// TIA Portal V17 export
// export: Created 2025-03-07T09:17:39.7845151Z, ExportSetting WithDefaults, DisplayName Totally Integrated Automation Portal, DisplayVersion V17 Update 8, DisplayName TIA Portal Openness, DisplayVersion V17 Update 8, DisplayName TIA Portal Version Control Interface, DisplayVersion V17, DisplayName SINAMICS Startdrive Advanced, DisplayVersion V17 SP2, DisplayName SINAMICS Startdrive G110M, G120, G120C, G120D, G120P, G115D, DisplayVersion V17 SP2, DisplayName SINAMICS Startdrive G130, G150, S120, S150, SINAMICS MV, S210, DisplayVersion V17 SP2, DisplayName STEP 7 Professional, DisplayVersion V17 Update 8, DisplayName SINUMERIK ONE STEP 7 Toolbox, DisplayVersion V17 Update 12, DisplayName SINUMERIK 840D sl STEP 7 Toolbox, DisplayVersion V17 Update 12, DisplayName STEP 7 Safety, DisplayVersion V17 Update 6, DisplayName WinCC Advanced, DisplayVersion V17 Update 8
FUNCTION "FC2001_AUTO_SINGLE_SEMI_MANUAL" : Void   // FC2001, LAD
{ S7_Optimized_Access := 'FALSE' }
AUTHOR : ETXETAR
VERSION : 1.0
// stored: AutoNumber false, IsIECCheckEnabled false, SetENOAutomatically false, UDAEnableTagReadback false
   VAR_TEMP
      O_BYTE_0 : Struct   // OPTIONS BYTE 0
         CHANGE_MODE_SEOC_ALARM : Bool;   // CHANGE MODE SEOC ALARM OPTION
         MODE_SELECTED_MEMORY : Bool;   // MODE SELECTED MEMORY OPTION
      END_STRUCT;
   END_VAR
   VAR CONSTANT
      FC_NUMBER : Int := 2001;   // NUMBER
   END_VAR
   VAR_TEMP   // added for the SCL form of the ladder/FBD networks
      _w1 : Bool;
      _w2 : Bool;
   END_VAR
BEGIN

REGION Network 1: OPTIONS OFF
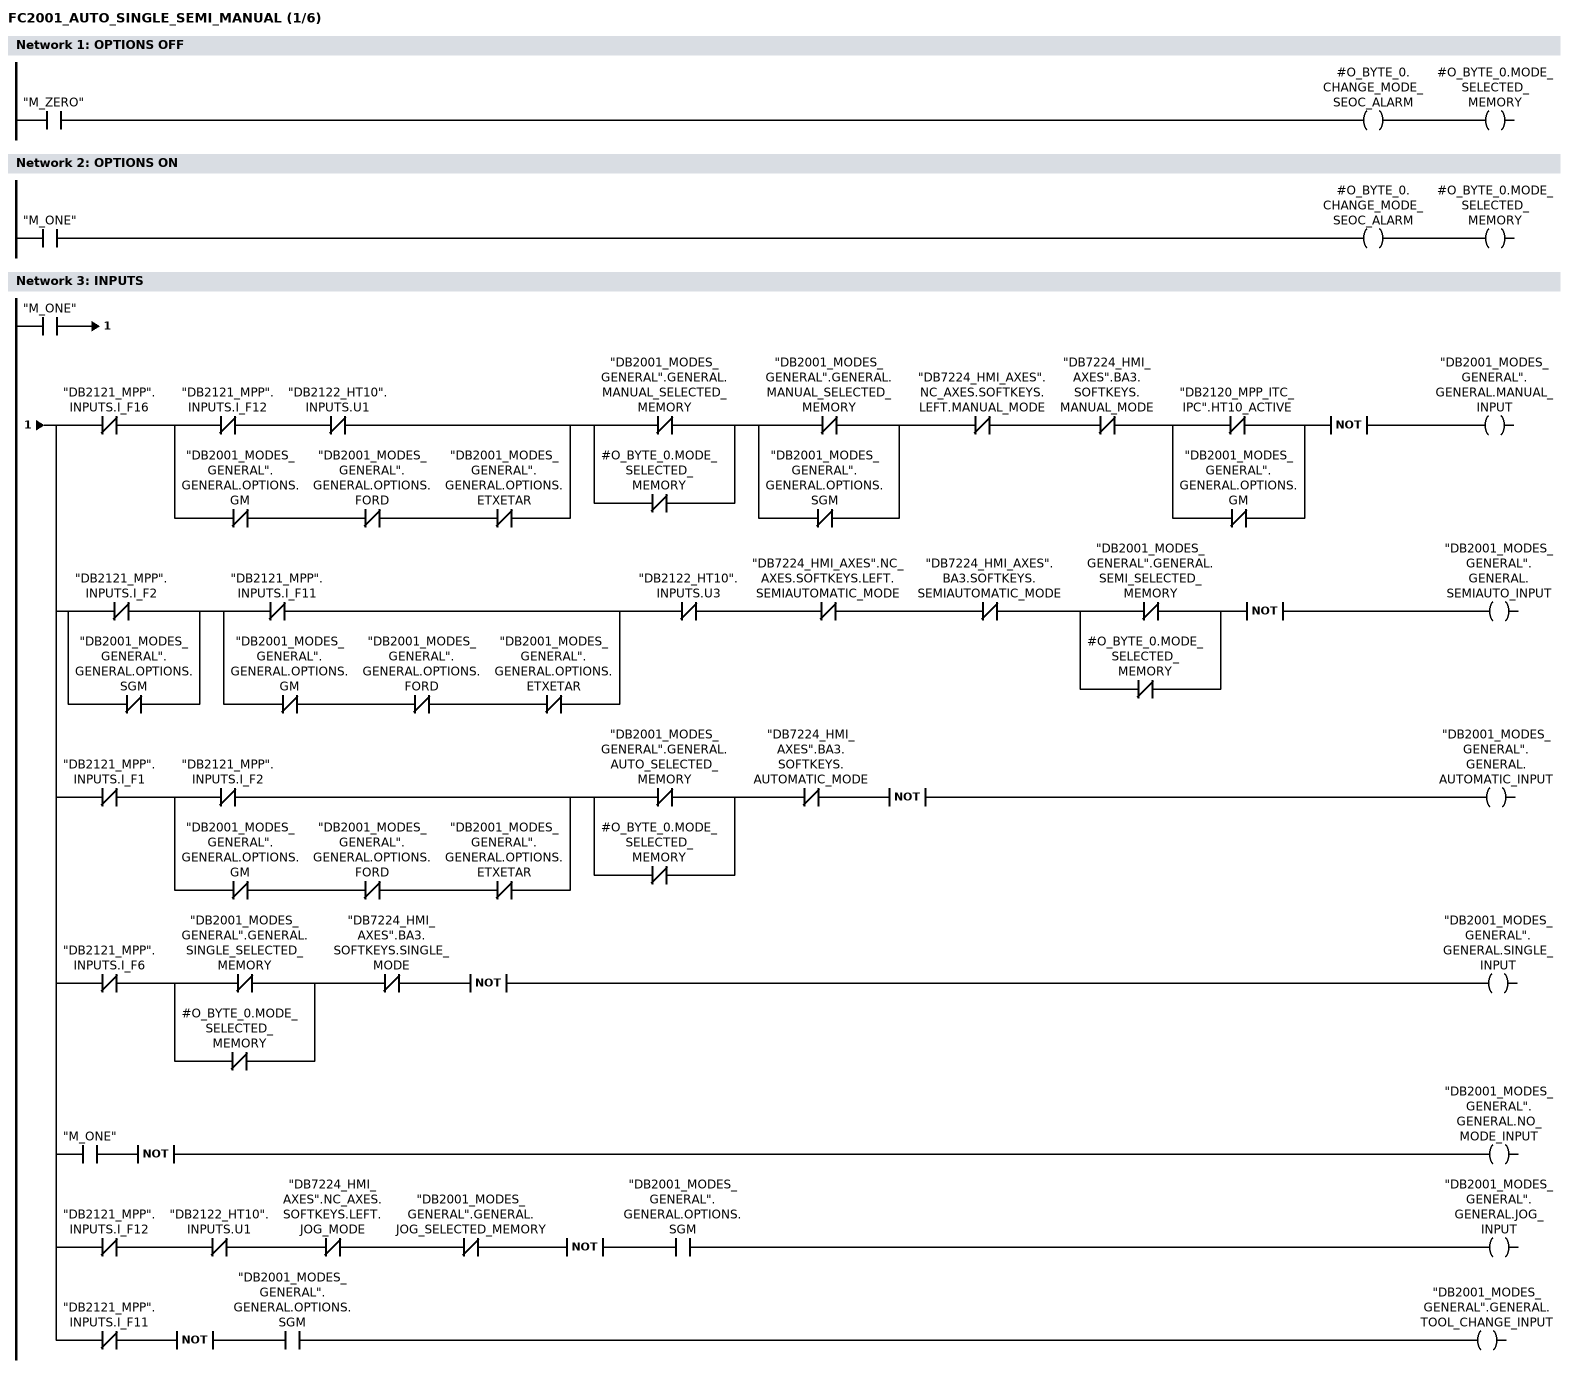
   RUNG wire#powerrail
      Contact( "M_ZERO" )
      Coil( #O_BYTE_0.CHANGE_MODE_SEOC_ALARM )
      Coil( #O_BYTE_0.MODE_SELECTED_MEMORY )
   END_RUNG
   // the same network as SCL:
   #O_BYTE_0.CHANGE_MODE_SEOC_ALARM := "M_ZERO";
   #O_BYTE_0.MODE_SELECTED_MEMORY := "M_ZERO";
END_REGION

REGION Network 2: OPTIONS ON
   RUNG wire#powerrail
      Contact( "M_ONE" )
      Coil( #O_BYTE_0.CHANGE_MODE_SEOC_ALARM )
      Coil( #O_BYTE_0.MODE_SELECTED_MEMORY )
   END_RUNG
   // the same network as SCL:
   #O_BYTE_0.CHANGE_MODE_SEOC_ALARM := "M_ONE";
   #O_BYTE_0.MODE_SELECTED_MEMORY := "M_ONE";
END_REGION

REGION Network 3: INPUTS
   RUNG wire#powerrail
      Contact( "M_ONE" )
      wire#w1
      I_Contact( "DB2121_MPP".INPUTS.I_F16 )
      wire#w2
      I_Contact( "DB2121_MPP".INPUTS.I_F12 )
      I_Contact( "DB2122_HT10".INPUTS.U1 )
      wire#w3
      I_Contact( "DB2001_MODES_GENERAL".GENERAL.MANUAL_SELECTED_MEMORY )
      wire#w4
      I_Contact( "DB2001_MODES_GENERAL".GENERAL.MANUAL_SELECTED_MEMORY )
      wire#w5
      I_Contact( "DB7224_HMI_AXES".NC_AXES.SOFTKEYS.LEFT.MANUAL_MODE )
      I_Contact( "DB7224_HMI_AXES".BA3.SOFTKEYS.MANUAL_MODE )
      wire#w6
      I_Contact( "DB2120_MPP_ITC_IPC".HT10_ACTIVE )
      wire#w7
      Not()
      Coil( "DB2001_MODES_GENERAL".GENERAL.MANUAL_INPUT )
   END_RUNG
   RUNG wire#w2
      I_Contact( "DB2001_MODES_GENERAL".GENERAL.OPTIONS.GM )
      I_Contact( "DB2001_MODES_GENERAL".GENERAL.OPTIONS.FORD )
      I_Contact( "DB2001_MODES_GENERAL".GENERAL.OPTIONS.ETXETAR )
   END_RUNG wire#w3
   RUNG wire#w3
      I_Contact( #O_BYTE_0.MODE_SELECTED_MEMORY )
   END_RUNG wire#w4
   RUNG wire#w4
      I_Contact( "DB2001_MODES_GENERAL".GENERAL.OPTIONS.SGM )
   END_RUNG wire#w5
   RUNG wire#w6
      I_Contact( "DB2001_MODES_GENERAL".GENERAL.OPTIONS.GM )
   END_RUNG wire#w7
   RUNG wire#w1
      I_Contact( "DB2121_MPP".INPUTS.I_F2 )
      wire#w8
      I_Contact( "DB2121_MPP".INPUTS.I_F11 )
      wire#w9
      I_Contact( "DB2122_HT10".INPUTS.U3 )
      I_Contact( "DB7224_HMI_AXES".NC_AXES.SOFTKEYS.LEFT.SEMIAUTOMATIC_MODE )
      I_Contact( "DB7224_HMI_AXES".BA3.SOFTKEYS.SEMIAUTOMATIC_MODE )
      wire#w10
      I_Contact( "DB2001_MODES_GENERAL".GENERAL.SEMI_SELECTED_MEMORY )
      wire#w11
      Not()
      Coil( "DB2001_MODES_GENERAL".GENERAL.SEMIAUTO_INPUT )
   END_RUNG
   RUNG wire#w1
      I_Contact( "DB2001_MODES_GENERAL".GENERAL.OPTIONS.SGM )
   END_RUNG wire#w8
   RUNG wire#w8
      I_Contact( "DB2001_MODES_GENERAL".GENERAL.OPTIONS.GM )
      I_Contact( "DB2001_MODES_GENERAL".GENERAL.OPTIONS.FORD )
      I_Contact( "DB2001_MODES_GENERAL".GENERAL.OPTIONS.ETXETAR )
   END_RUNG wire#w9
   RUNG wire#w10
      I_Contact( #O_BYTE_0.MODE_SELECTED_MEMORY )
   END_RUNG wire#w11
   RUNG wire#w1
      I_Contact( "DB2121_MPP".INPUTS.I_F1 )
      wire#w12
      I_Contact( "DB2121_MPP".INPUTS.I_F2 )
      wire#w13
      I_Contact( "DB2001_MODES_GENERAL".GENERAL.AUTO_SELECTED_MEMORY )
      wire#w14
      I_Contact( "DB7224_HMI_AXES".BA3.SOFTKEYS.AUTOMATIC_MODE )
      Not()
      Coil( "DB2001_MODES_GENERAL".GENERAL.AUTOMATIC_INPUT )
   END_RUNG
   RUNG wire#w12
      I_Contact( "DB2001_MODES_GENERAL".GENERAL.OPTIONS.GM )
      I_Contact( "DB2001_MODES_GENERAL".GENERAL.OPTIONS.FORD )
      I_Contact( "DB2001_MODES_GENERAL".GENERAL.OPTIONS.ETXETAR )
   END_RUNG wire#w13
   RUNG wire#w13
      I_Contact( #O_BYTE_0.MODE_SELECTED_MEMORY )
   END_RUNG wire#w14
   RUNG wire#w1
      I_Contact( "DB2121_MPP".INPUTS.I_F6 )
      wire#w15
      I_Contact( "DB2001_MODES_GENERAL".GENERAL.SINGLE_SELECTED_MEMORY )
      wire#w16
      I_Contact( "DB7224_HMI_AXES".BA3.SOFTKEYS.SINGLE_MODE )
      Not()
      Coil( "DB2001_MODES_GENERAL".GENERAL.SINGLE_INPUT )
   END_RUNG
   RUNG wire#w15
      I_Contact( #O_BYTE_0.MODE_SELECTED_MEMORY )
   END_RUNG wire#w16
   RUNG wire#w1
      Contact( "M_ONE" )
      Not()
      Coil( "DB2001_MODES_GENERAL".GENERAL.NO_MODE_INPUT )
   END_RUNG
   RUNG wire#w1
      I_Contact( "DB2121_MPP".INPUTS.I_F12 )
      I_Contact( "DB2122_HT10".INPUTS.U1 )
      I_Contact( "DB7224_HMI_AXES".NC_AXES.SOFTKEYS.LEFT.JOG_MODE )
      I_Contact( "DB2001_MODES_GENERAL".GENERAL.JOG_SELECTED_MEMORY )
      Not()
      Contact( "DB2001_MODES_GENERAL".GENERAL.OPTIONS.SGM )
      Coil( "DB2001_MODES_GENERAL".GENERAL.JOG_INPUT )
   END_RUNG
   RUNG wire#w1
      I_Contact( "DB2121_MPP".INPUTS.I_F11 )
      Not()
      Contact( "DB2001_MODES_GENERAL".GENERAL.OPTIONS.SGM )
      Coil( "DB2001_MODES_GENERAL".GENERAL.TOOL_CHANGE_INPUT )
   END_RUNG
   // the same network as SCL:
   "DB2001_MODES_GENERAL".GENERAL.MANUAL_INPUT := NOT ("M_ONE" AND NOT "DB2121_MPP".INPUTS.I_F16 AND ((NOT "DB2121_MPP".INPUTS.I_F12 AND NOT "DB2122_HT10".INPUTS.U1) OR (NOT "DB2001_MODES_GENERAL".GENERAL.OPTIONS.GM AND NOT "DB2001_MODES_GENERAL".GENERAL.OPTIONS.FORD AND NOT "DB2001_MODES_GENERAL".GENERAL.OPTIONS.ETXETAR)) AND (NOT "DB2001_MODES_GENERAL".GENERAL.MANUAL_SELECTED_MEMORY OR NOT #O_BYTE_0.MODE_SELECTED_MEMORY) AND (NOT "DB2001_MODES_GENERAL".GENERAL.MANUAL_SELECTED_MEMORY OR NOT "DB2001_MODES_GENERAL".GENERAL.OPTIONS.SGM) AND NOT "DB7224_HMI_AXES".NC_AXES.SOFTKEYS.LEFT.MANUAL_MODE AND NOT "DB7224_HMI_AXES".BA3.SOFTKEYS.MANUAL_MODE AND (NOT "DB2120_MPP_ITC_IPC".HT10_ACTIVE OR NOT "DB2001_MODES_GENERAL".GENERAL.OPTIONS.GM));
   "DB2001_MODES_GENERAL".GENERAL.SEMIAUTO_INPUT := NOT ("M_ONE" AND (NOT "DB2121_MPP".INPUTS.I_F2 OR NOT "DB2001_MODES_GENERAL".GENERAL.OPTIONS.SGM) AND (NOT "DB2121_MPP".INPUTS.I_F11 OR (NOT "DB2001_MODES_GENERAL".GENERAL.OPTIONS.GM AND NOT "DB2001_MODES_GENERAL".GENERAL.OPTIONS.FORD AND NOT "DB2001_MODES_GENERAL".GENERAL.OPTIONS.ETXETAR)) AND NOT "DB2122_HT10".INPUTS.U3 AND NOT "DB7224_HMI_AXES".NC_AXES.SOFTKEYS.LEFT.SEMIAUTOMATIC_MODE AND NOT "DB7224_HMI_AXES".BA3.SOFTKEYS.SEMIAUTOMATIC_MODE AND (NOT "DB2001_MODES_GENERAL".GENERAL.SEMI_SELECTED_MEMORY OR NOT #O_BYTE_0.MODE_SELECTED_MEMORY));
   "DB2001_MODES_GENERAL".GENERAL.AUTOMATIC_INPUT := NOT ("M_ONE" AND NOT "DB2121_MPP".INPUTS.I_F1 AND (NOT "DB2121_MPP".INPUTS.I_F2 OR (NOT "DB2001_MODES_GENERAL".GENERAL.OPTIONS.GM AND NOT "DB2001_MODES_GENERAL".GENERAL.OPTIONS.FORD AND NOT "DB2001_MODES_GENERAL".GENERAL.OPTIONS.ETXETAR)) AND (NOT "DB2001_MODES_GENERAL".GENERAL.AUTO_SELECTED_MEMORY OR NOT #O_BYTE_0.MODE_SELECTED_MEMORY) AND NOT "DB7224_HMI_AXES".BA3.SOFTKEYS.AUTOMATIC_MODE);
   "DB2001_MODES_GENERAL".GENERAL.SINGLE_INPUT := NOT ("M_ONE" AND NOT "DB2121_MPP".INPUTS.I_F6 AND (NOT "DB2001_MODES_GENERAL".GENERAL.SINGLE_SELECTED_MEMORY OR NOT #O_BYTE_0.MODE_SELECTED_MEMORY) AND NOT "DB7224_HMI_AXES".BA3.SOFTKEYS.SINGLE_MODE);
   "DB2001_MODES_GENERAL".GENERAL.NO_MODE_INPUT := NOT ("M_ONE" AND "M_ONE");
   "DB2001_MODES_GENERAL".GENERAL.JOG_INPUT := NOT ("M_ONE" AND NOT "DB2121_MPP".INPUTS.I_F12 AND NOT "DB2122_HT10".INPUTS.U1 AND NOT "DB7224_HMI_AXES".NC_AXES.SOFTKEYS.LEFT.JOG_MODE AND NOT "DB2001_MODES_GENERAL".GENERAL.JOG_SELECTED_MEMORY) AND "DB2001_MODES_GENERAL".GENERAL.OPTIONS.SGM;
   "DB2001_MODES_GENERAL".GENERAL.TOOL_CHANGE_INPUT := NOT ("M_ONE" AND NOT "DB2121_MPP".INPUTS.I_F11) AND "DB2001_MODES_GENERAL".GENERAL.OPTIONS.SGM;
END_REGION

REGION Network 4: SGM CHANGE MODE MEMORIES
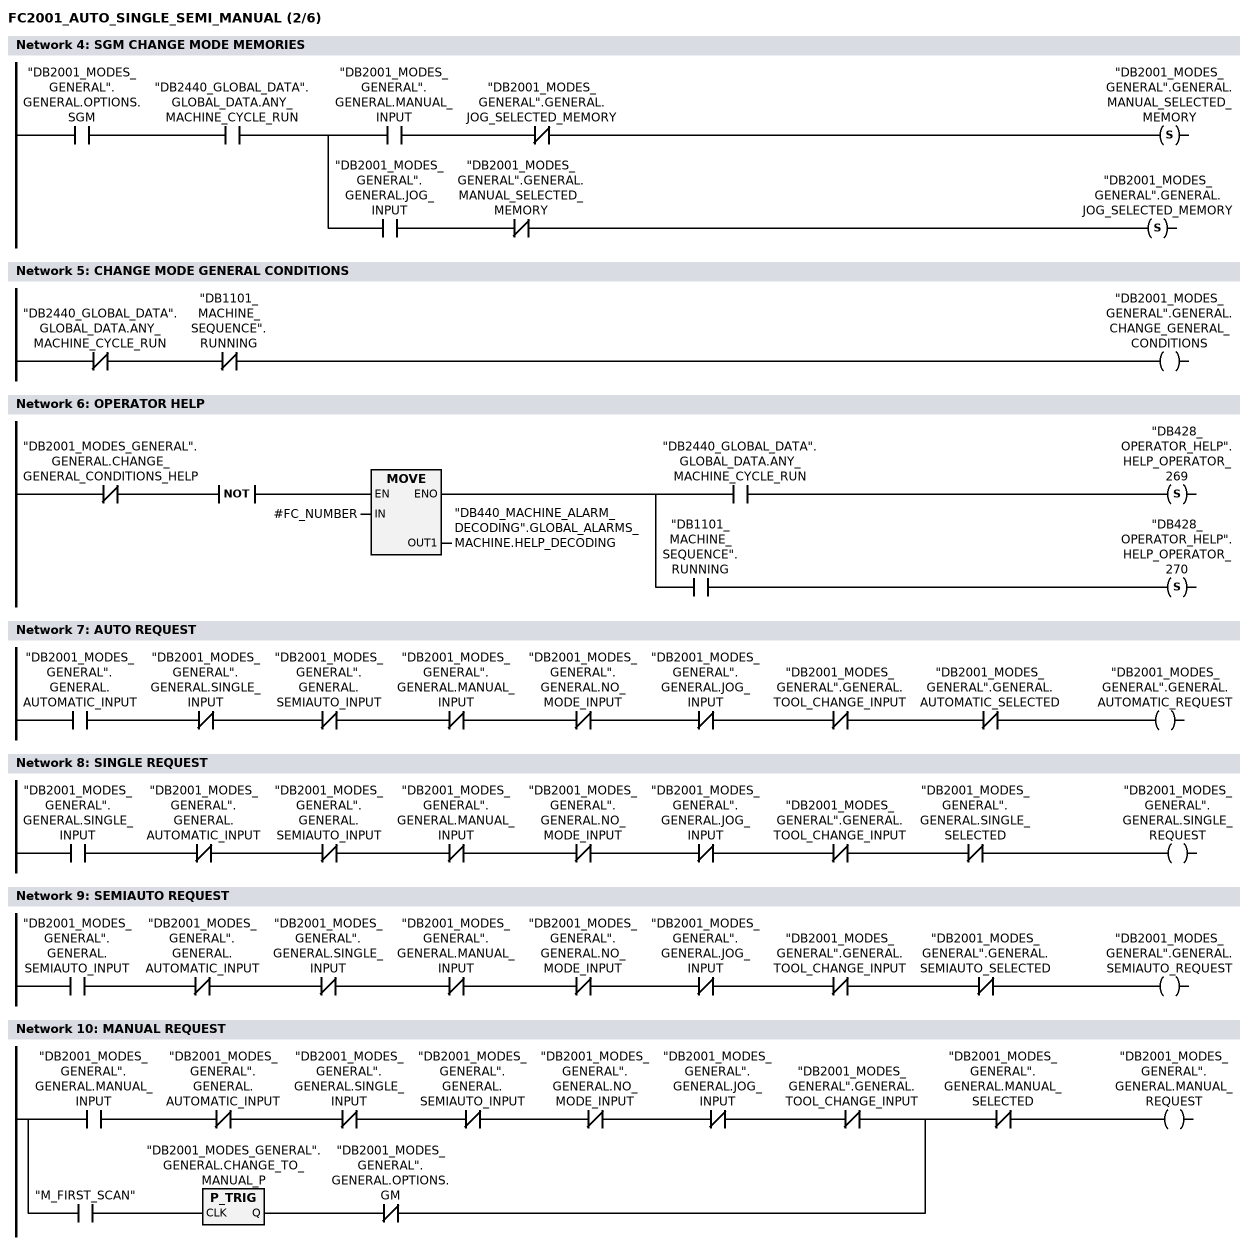
   RUNG wire#powerrail
      Contact( "DB2001_MODES_GENERAL".GENERAL.OPTIONS.SGM )
      Contact( "DB2440_GLOBAL_DATA".GLOBAL_DATA.ANY_MACHINE_CYCLE_RUN )
      wire#w1
      Contact( "DB2001_MODES_GENERAL".GENERAL.MANUAL_INPUT )
      I_Contact( "DB2001_MODES_GENERAL".GENERAL.JOG_SELECTED_MEMORY )
      S_Coil( "DB2001_MODES_GENERAL".GENERAL.MANUAL_SELECTED_MEMORY )
   END_RUNG
   RUNG wire#w1
      Contact( "DB2001_MODES_GENERAL".GENERAL.JOG_INPUT )
      I_Contact( "DB2001_MODES_GENERAL".GENERAL.MANUAL_SELECTED_MEMORY )
      S_Coil( "DB2001_MODES_GENERAL".GENERAL.JOG_SELECTED_MEMORY )
   END_RUNG
   // the same network as SCL:
   #_w1 := "DB2001_MODES_GENERAL".GENERAL.OPTIONS.SGM AND "DB2440_GLOBAL_DATA".GLOBAL_DATA.ANY_MACHINE_CYCLE_RUN;
   IF #_w1 AND "DB2001_MODES_GENERAL".GENERAL.MANUAL_INPUT AND NOT "DB2001_MODES_GENERAL".GENERAL.JOG_SELECTED_MEMORY THEN
       "DB2001_MODES_GENERAL".GENERAL.MANUAL_SELECTED_MEMORY := TRUE;
   END_IF;
   IF #_w1 AND "DB2001_MODES_GENERAL".GENERAL.JOG_INPUT AND NOT "DB2001_MODES_GENERAL".GENERAL.MANUAL_SELECTED_MEMORY THEN
       "DB2001_MODES_GENERAL".GENERAL.JOG_SELECTED_MEMORY := TRUE;
   END_IF;
END_REGION

REGION Network 5: CHANGE MODE GENERAL CONDITIONS
   RUNG wire#powerrail
      I_Contact( "DB2440_GLOBAL_DATA".GLOBAL_DATA.ANY_MACHINE_CYCLE_RUN )
      I_Contact( "DB1101_MACHINE_SEQUENCE".RUNNING )
      Coil( "DB2001_MODES_GENERAL".GENERAL.CHANGE_GENERAL_CONDITIONS )
   END_RUNG
   // the same network as SCL:
   "DB2001_MODES_GENERAL".GENERAL.CHANGE_GENERAL_CONDITIONS := NOT "DB2440_GLOBAL_DATA".GLOBAL_DATA.ANY_MACHINE_CYCLE_RUN AND NOT "DB1101_MACHINE_SEQUENCE".RUNNING;
END_REGION

REGION Network 6: OPERATOR HELP
   RUNG wire#powerrail
      I_Contact( "DB2001_MODES_GENERAL".GENERAL.CHANGE_GENERAL_CONDITIONS_HELP )
      Not()
      { S7_GenerateENO := "TRUE" } Move(in := #FC_NUMBER, out1 => "DB440_MACHINE_ALARM_DECODING".GLOBAL_ALARMS_MACHINE.HELP_DECODING)
      wire#w1
      Contact( "DB2440_GLOBAL_DATA".GLOBAL_DATA.ANY_MACHINE_CYCLE_RUN )
      S_Coil( "DB428_OPERATOR_HELP".HELP_OPERATOR_269 )
   END_RUNG
   RUNG wire#w1
      Contact( "DB1101_MACHINE_SEQUENCE".RUNNING )
      S_Coil( "DB428_OPERATOR_HELP".HELP_OPERATOR_270 )
   END_RUNG
   // the same network as SCL:
   // ENO of a box is taken as its EN; it also drops when the box reports an error
   #_w1 := NOT (NOT "DB2001_MODES_GENERAL".GENERAL.CHANGE_GENERAL_CONDITIONS_HELP);
   IF #_w1 THEN "DB440_MACHINE_ALARM_DECODING".GLOBAL_ALARMS_MACHINE.HELP_DECODING := #FC_NUMBER; END_IF;
   IF #_w1 AND "DB2440_GLOBAL_DATA".GLOBAL_DATA.ANY_MACHINE_CYCLE_RUN THEN
       "DB428_OPERATOR_HELP".HELP_OPERATOR_269 := TRUE;
   END_IF;
   IF #_w1 AND "DB1101_MACHINE_SEQUENCE".RUNNING THEN
       "DB428_OPERATOR_HELP".HELP_OPERATOR_270 := TRUE;
   END_IF;
END_REGION

REGION Network 7: AUTO REQUEST
   RUNG wire#powerrail
      Contact( "DB2001_MODES_GENERAL".GENERAL.AUTOMATIC_INPUT )
      I_Contact( "DB2001_MODES_GENERAL".GENERAL.SINGLE_INPUT )
      I_Contact( "DB2001_MODES_GENERAL".GENERAL.SEMIAUTO_INPUT )
      I_Contact( "DB2001_MODES_GENERAL".GENERAL.MANUAL_INPUT )
      I_Contact( "DB2001_MODES_GENERAL".GENERAL.NO_MODE_INPUT )
      I_Contact( "DB2001_MODES_GENERAL".GENERAL.JOG_INPUT )
      I_Contact( "DB2001_MODES_GENERAL".GENERAL.TOOL_CHANGE_INPUT )
      I_Contact( "DB2001_MODES_GENERAL".GENERAL.AUTOMATIC_SELECTED )
      Coil( "DB2001_MODES_GENERAL".GENERAL.AUTOMATIC_REQUEST )
   END_RUNG
   // the same network as SCL:
   "DB2001_MODES_GENERAL".GENERAL.AUTOMATIC_REQUEST := "DB2001_MODES_GENERAL".GENERAL.AUTOMATIC_INPUT AND NOT "DB2001_MODES_GENERAL".GENERAL.SINGLE_INPUT AND NOT "DB2001_MODES_GENERAL".GENERAL.SEMIAUTO_INPUT AND NOT "DB2001_MODES_GENERAL".GENERAL.MANUAL_INPUT AND NOT "DB2001_MODES_GENERAL".GENERAL.NO_MODE_INPUT AND NOT "DB2001_MODES_GENERAL".GENERAL.JOG_INPUT AND NOT "DB2001_MODES_GENERAL".GENERAL.TOOL_CHANGE_INPUT AND NOT "DB2001_MODES_GENERAL".GENERAL.AUTOMATIC_SELECTED;
END_REGION

REGION Network 8: SINGLE REQUEST
   RUNG wire#powerrail
      Contact( "DB2001_MODES_GENERAL".GENERAL.SINGLE_INPUT )
      I_Contact( "DB2001_MODES_GENERAL".GENERAL.AUTOMATIC_INPUT )
      I_Contact( "DB2001_MODES_GENERAL".GENERAL.SEMIAUTO_INPUT )
      I_Contact( "DB2001_MODES_GENERAL".GENERAL.MANUAL_INPUT )
      I_Contact( "DB2001_MODES_GENERAL".GENERAL.NO_MODE_INPUT )
      I_Contact( "DB2001_MODES_GENERAL".GENERAL.JOG_INPUT )
      I_Contact( "DB2001_MODES_GENERAL".GENERAL.TOOL_CHANGE_INPUT )
      I_Contact( "DB2001_MODES_GENERAL".GENERAL.SINGLE_SELECTED )
      Coil( "DB2001_MODES_GENERAL".GENERAL.SINGLE_REQUEST )
   END_RUNG
   // the same network as SCL:
   "DB2001_MODES_GENERAL".GENERAL.SINGLE_REQUEST := "DB2001_MODES_GENERAL".GENERAL.SINGLE_INPUT AND NOT "DB2001_MODES_GENERAL".GENERAL.AUTOMATIC_INPUT AND NOT "DB2001_MODES_GENERAL".GENERAL.SEMIAUTO_INPUT AND NOT "DB2001_MODES_GENERAL".GENERAL.MANUAL_INPUT AND NOT "DB2001_MODES_GENERAL".GENERAL.NO_MODE_INPUT AND NOT "DB2001_MODES_GENERAL".GENERAL.JOG_INPUT AND NOT "DB2001_MODES_GENERAL".GENERAL.TOOL_CHANGE_INPUT AND NOT "DB2001_MODES_GENERAL".GENERAL.SINGLE_SELECTED;
END_REGION

REGION Network 9: SEMIAUTO REQUEST
   RUNG wire#powerrail
      Contact( "DB2001_MODES_GENERAL".GENERAL.SEMIAUTO_INPUT )
      I_Contact( "DB2001_MODES_GENERAL".GENERAL.AUTOMATIC_INPUT )
      I_Contact( "DB2001_MODES_GENERAL".GENERAL.SINGLE_INPUT )
      I_Contact( "DB2001_MODES_GENERAL".GENERAL.MANUAL_INPUT )
      I_Contact( "DB2001_MODES_GENERAL".GENERAL.NO_MODE_INPUT )
      I_Contact( "DB2001_MODES_GENERAL".GENERAL.JOG_INPUT )
      I_Contact( "DB2001_MODES_GENERAL".GENERAL.TOOL_CHANGE_INPUT )
      I_Contact( "DB2001_MODES_GENERAL".GENERAL.SEMIAUTO_SELECTED )
      Coil( "DB2001_MODES_GENERAL".GENERAL.SEMIAUTO_REQUEST )
   END_RUNG
   // the same network as SCL:
   "DB2001_MODES_GENERAL".GENERAL.SEMIAUTO_REQUEST := "DB2001_MODES_GENERAL".GENERAL.SEMIAUTO_INPUT AND NOT "DB2001_MODES_GENERAL".GENERAL.AUTOMATIC_INPUT AND NOT "DB2001_MODES_GENERAL".GENERAL.SINGLE_INPUT AND NOT "DB2001_MODES_GENERAL".GENERAL.MANUAL_INPUT AND NOT "DB2001_MODES_GENERAL".GENERAL.NO_MODE_INPUT AND NOT "DB2001_MODES_GENERAL".GENERAL.JOG_INPUT AND NOT "DB2001_MODES_GENERAL".GENERAL.TOOL_CHANGE_INPUT AND NOT "DB2001_MODES_GENERAL".GENERAL.SEMIAUTO_SELECTED;
END_REGION

REGION Network 10: MANUAL REQUEST
   RUNG wire#powerrail
      Contact( "DB2001_MODES_GENERAL".GENERAL.MANUAL_INPUT )
      I_Contact( "DB2001_MODES_GENERAL".GENERAL.AUTOMATIC_INPUT )
      I_Contact( "DB2001_MODES_GENERAL".GENERAL.SINGLE_INPUT )
      I_Contact( "DB2001_MODES_GENERAL".GENERAL.SEMIAUTO_INPUT )
      I_Contact( "DB2001_MODES_GENERAL".GENERAL.NO_MODE_INPUT )
      I_Contact( "DB2001_MODES_GENERAL".GENERAL.JOG_INPUT )
      I_Contact( "DB2001_MODES_GENERAL".GENERAL.TOOL_CHANGE_INPUT )
      wire#w1
      I_Contact( "DB2001_MODES_GENERAL".GENERAL.MANUAL_SELECTED )
      Coil( "DB2001_MODES_GENERAL".GENERAL.MANUAL_REQUEST )
   END_RUNG
   RUNG wire#powerrail
      Contact( "M_FIRST_SCAN" )
      P_Trig( "DB2001_MODES_GENERAL".GENERAL.CHANGE_TO_MANUAL_P )
      I_Contact( "DB2001_MODES_GENERAL".GENERAL.OPTIONS.GM )
   END_RUNG wire#w1
   // the same network as SCL:
   #_w1 := "M_FIRST_SCAN" AND NOT "DB2001_MODES_GENERAL".GENERAL.CHANGE_TO_MANUAL_P;   // rising edge
   "DB2001_MODES_GENERAL".GENERAL.CHANGE_TO_MANUAL_P := "M_FIRST_SCAN";
   "DB2001_MODES_GENERAL".GENERAL.MANUAL_REQUEST := (("DB2001_MODES_GENERAL".GENERAL.MANUAL_INPUT AND NOT "DB2001_MODES_GENERAL".GENERAL.AUTOMATIC_INPUT AND NOT "DB2001_MODES_GENERAL".GENERAL.SINGLE_INPUT AND NOT "DB2001_MODES_GENERAL".GENERAL.SEMIAUTO_INPUT AND NOT "DB2001_MODES_GENERAL".GENERAL.NO_MODE_INPUT AND NOT "DB2001_MODES_GENERAL".GENERAL.JOG_INPUT AND NOT "DB2001_MODES_GENERAL".GENERAL.TOOL_CHANGE_INPUT) OR (#_w1 AND NOT "DB2001_MODES_GENERAL".GENERAL.OPTIONS.GM)) AND NOT "DB2001_MODES_GENERAL".GENERAL.MANUAL_SELECTED;
END_REGION

REGION Network 11: NO MODE REQUEST
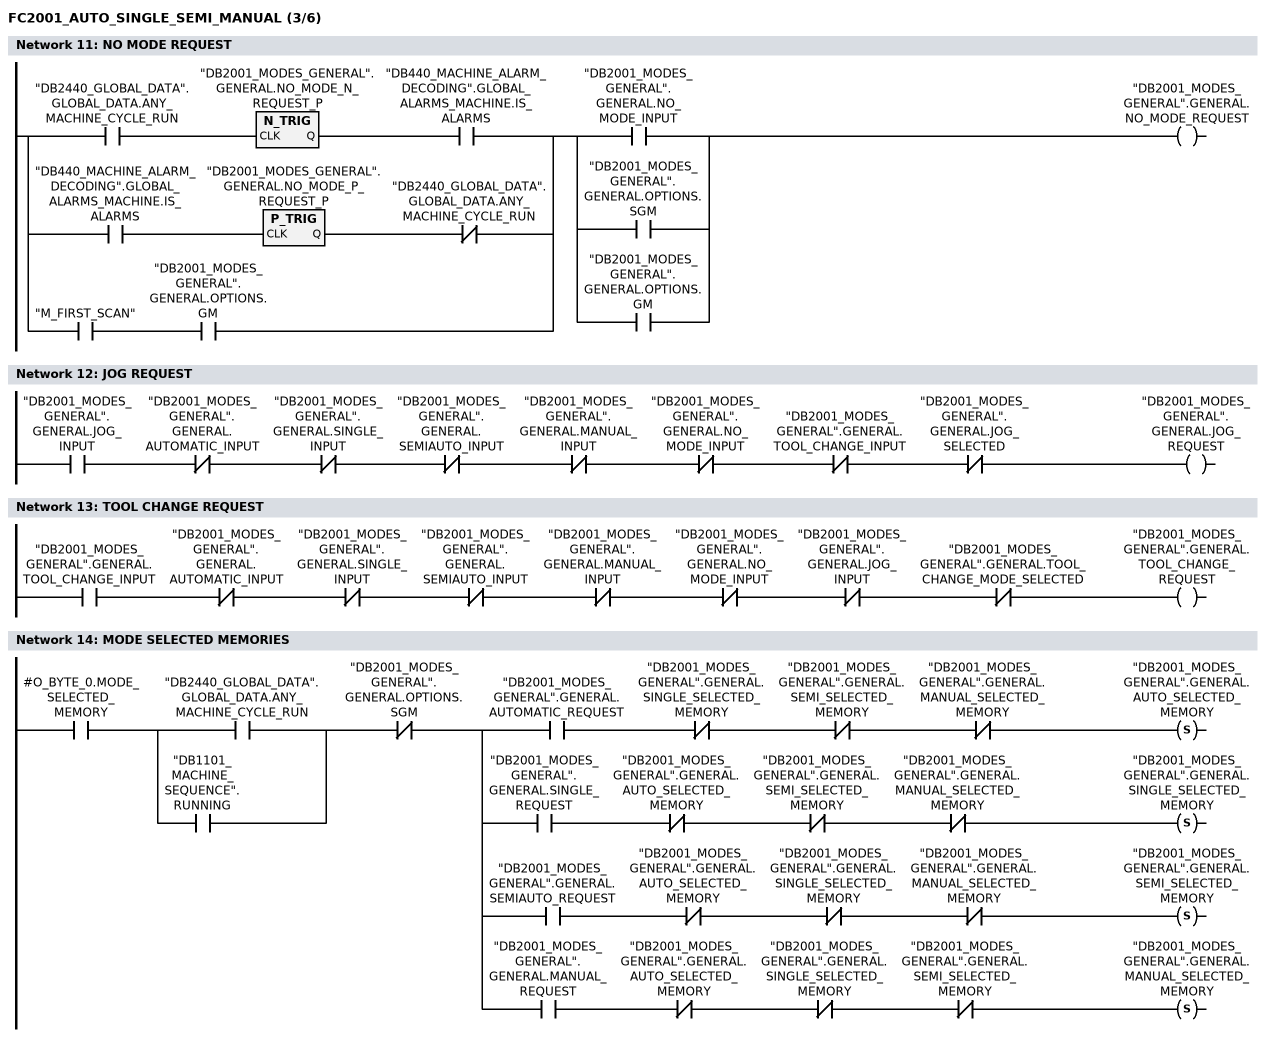
   RUNG wire#powerrail
      Contact( "DB2440_GLOBAL_DATA".GLOBAL_DATA.ANY_MACHINE_CYCLE_RUN )
      N_Trig( "DB2001_MODES_GENERAL".GENERAL.NO_MODE_N_REQUEST_P )
      Contact( "DB440_MACHINE_ALARM_DECODING".GLOBAL_ALARMS_MACHINE.IS_ALARMS )
      wire#w1
      Contact( "DB2001_MODES_GENERAL".GENERAL.NO_MODE_INPUT )
      wire#w2
      Coil( "DB2001_MODES_GENERAL".GENERAL.NO_MODE_REQUEST )
   END_RUNG
   RUNG wire#powerrail
      Contact( "DB440_MACHINE_ALARM_DECODING".GLOBAL_ALARMS_MACHINE.IS_ALARMS )
      P_Trig( "DB2001_MODES_GENERAL".GENERAL.NO_MODE_P_REQUEST_P )
      I_Contact( "DB2440_GLOBAL_DATA".GLOBAL_DATA.ANY_MACHINE_CYCLE_RUN )
   END_RUNG wire#w1
   RUNG wire#powerrail
      Contact( "M_FIRST_SCAN" )
      Contact( "DB2001_MODES_GENERAL".GENERAL.OPTIONS.GM )
   END_RUNG wire#w1
   RUNG wire#w1
      Contact( "DB2001_MODES_GENERAL".GENERAL.OPTIONS.SGM )
   END_RUNG wire#w2
   RUNG wire#w1
      Contact( "DB2001_MODES_GENERAL".GENERAL.OPTIONS.GM )
   END_RUNG wire#w2
   // the same network as SCL:
   #_w1 := NOT "DB2440_GLOBAL_DATA".GLOBAL_DATA.ANY_MACHINE_CYCLE_RUN AND "DB2001_MODES_GENERAL".GENERAL.NO_MODE_N_REQUEST_P;   // falling edge
   "DB2001_MODES_GENERAL".GENERAL.NO_MODE_N_REQUEST_P := "DB2440_GLOBAL_DATA".GLOBAL_DATA.ANY_MACHINE_CYCLE_RUN;
   #_w2 := "DB440_MACHINE_ALARM_DECODING".GLOBAL_ALARMS_MACHINE.IS_ALARMS AND NOT "DB2001_MODES_GENERAL".GENERAL.NO_MODE_P_REQUEST_P;   // rising edge
   "DB2001_MODES_GENERAL".GENERAL.NO_MODE_P_REQUEST_P := "DB440_MACHINE_ALARM_DECODING".GLOBAL_ALARMS_MACHINE.IS_ALARMS;
   "DB2001_MODES_GENERAL".GENERAL.NO_MODE_REQUEST := ((#_w1 AND "DB440_MACHINE_ALARM_DECODING".GLOBAL_ALARMS_MACHINE.IS_ALARMS) OR (#_w2 AND NOT "DB2440_GLOBAL_DATA".GLOBAL_DATA.ANY_MACHINE_CYCLE_RUN) OR ("M_FIRST_SCAN" AND "DB2001_MODES_GENERAL".GENERAL.OPTIONS.GM)) AND ("DB2001_MODES_GENERAL".GENERAL.NO_MODE_INPUT OR "DB2001_MODES_GENERAL".GENERAL.OPTIONS.SGM OR "DB2001_MODES_GENERAL".GENERAL.OPTIONS.GM);
END_REGION

REGION Network 12: JOG REQUEST
   RUNG wire#powerrail
      Contact( "DB2001_MODES_GENERAL".GENERAL.JOG_INPUT )
      I_Contact( "DB2001_MODES_GENERAL".GENERAL.AUTOMATIC_INPUT )
      I_Contact( "DB2001_MODES_GENERAL".GENERAL.SINGLE_INPUT )
      I_Contact( "DB2001_MODES_GENERAL".GENERAL.SEMIAUTO_INPUT )
      I_Contact( "DB2001_MODES_GENERAL".GENERAL.MANUAL_INPUT )
      I_Contact( "DB2001_MODES_GENERAL".GENERAL.NO_MODE_INPUT )
      I_Contact( "DB2001_MODES_GENERAL".GENERAL.TOOL_CHANGE_INPUT )
      I_Contact( "DB2001_MODES_GENERAL".GENERAL.JOG_SELECTED )
      Coil( "DB2001_MODES_GENERAL".GENERAL.JOG_REQUEST )
   END_RUNG
   // the same network as SCL:
   "DB2001_MODES_GENERAL".GENERAL.JOG_REQUEST := "DB2001_MODES_GENERAL".GENERAL.JOG_INPUT AND NOT "DB2001_MODES_GENERAL".GENERAL.AUTOMATIC_INPUT AND NOT "DB2001_MODES_GENERAL".GENERAL.SINGLE_INPUT AND NOT "DB2001_MODES_GENERAL".GENERAL.SEMIAUTO_INPUT AND NOT "DB2001_MODES_GENERAL".GENERAL.MANUAL_INPUT AND NOT "DB2001_MODES_GENERAL".GENERAL.NO_MODE_INPUT AND NOT "DB2001_MODES_GENERAL".GENERAL.TOOL_CHANGE_INPUT AND NOT "DB2001_MODES_GENERAL".GENERAL.JOG_SELECTED;
END_REGION

REGION Network 13: TOOL CHANGE REQUEST
   RUNG wire#powerrail
      Contact( "DB2001_MODES_GENERAL".GENERAL.TOOL_CHANGE_INPUT )
      I_Contact( "DB2001_MODES_GENERAL".GENERAL.AUTOMATIC_INPUT )
      I_Contact( "DB2001_MODES_GENERAL".GENERAL.SINGLE_INPUT )
      I_Contact( "DB2001_MODES_GENERAL".GENERAL.SEMIAUTO_INPUT )
      I_Contact( "DB2001_MODES_GENERAL".GENERAL.MANUAL_INPUT )
      I_Contact( "DB2001_MODES_GENERAL".GENERAL.NO_MODE_INPUT )
      I_Contact( "DB2001_MODES_GENERAL".GENERAL.JOG_INPUT )
      I_Contact( "DB2001_MODES_GENERAL".GENERAL.TOOL_CHANGE_MODE_SELECTED )
      Coil( "DB2001_MODES_GENERAL".GENERAL.TOOL_CHANGE_REQUEST )
   END_RUNG
   // the same network as SCL:
   "DB2001_MODES_GENERAL".GENERAL.TOOL_CHANGE_REQUEST := "DB2001_MODES_GENERAL".GENERAL.TOOL_CHANGE_INPUT AND NOT "DB2001_MODES_GENERAL".GENERAL.AUTOMATIC_INPUT AND NOT "DB2001_MODES_GENERAL".GENERAL.SINGLE_INPUT AND NOT "DB2001_MODES_GENERAL".GENERAL.SEMIAUTO_INPUT AND NOT "DB2001_MODES_GENERAL".GENERAL.MANUAL_INPUT AND NOT "DB2001_MODES_GENERAL".GENERAL.NO_MODE_INPUT AND NOT "DB2001_MODES_GENERAL".GENERAL.JOG_INPUT AND NOT "DB2001_MODES_GENERAL".GENERAL.TOOL_CHANGE_MODE_SELECTED;
END_REGION

REGION Network 14: MODE SELECTED MEMORIES
   RUNG wire#powerrail
      Contact( #O_BYTE_0.MODE_SELECTED_MEMORY )
      wire#w1
      Contact( "DB2440_GLOBAL_DATA".GLOBAL_DATA.ANY_MACHINE_CYCLE_RUN )
      wire#w2
      I_Contact( "DB2001_MODES_GENERAL".GENERAL.OPTIONS.SGM )
      wire#w3
      Contact( "DB2001_MODES_GENERAL".GENERAL.AUTOMATIC_REQUEST )
      I_Contact( "DB2001_MODES_GENERAL".GENERAL.SINGLE_SELECTED_MEMORY )
      I_Contact( "DB2001_MODES_GENERAL".GENERAL.SEMI_SELECTED_MEMORY )
      I_Contact( "DB2001_MODES_GENERAL".GENERAL.MANUAL_SELECTED_MEMORY )
      S_Coil( "DB2001_MODES_GENERAL".GENERAL.AUTO_SELECTED_MEMORY )
   END_RUNG
   RUNG wire#w1
      Contact( "DB1101_MACHINE_SEQUENCE".RUNNING )
   END_RUNG wire#w2
   RUNG wire#w3
      Contact( "DB2001_MODES_GENERAL".GENERAL.SINGLE_REQUEST )
      I_Contact( "DB2001_MODES_GENERAL".GENERAL.AUTO_SELECTED_MEMORY )
      I_Contact( "DB2001_MODES_GENERAL".GENERAL.SEMI_SELECTED_MEMORY )
      I_Contact( "DB2001_MODES_GENERAL".GENERAL.MANUAL_SELECTED_MEMORY )
      S_Coil( "DB2001_MODES_GENERAL".GENERAL.SINGLE_SELECTED_MEMORY )
   END_RUNG
   RUNG wire#w3
      Contact( "DB2001_MODES_GENERAL".GENERAL.SEMIAUTO_REQUEST )
      I_Contact( "DB2001_MODES_GENERAL".GENERAL.AUTO_SELECTED_MEMORY )
      I_Contact( "DB2001_MODES_GENERAL".GENERAL.SINGLE_SELECTED_MEMORY )
      I_Contact( "DB2001_MODES_GENERAL".GENERAL.MANUAL_SELECTED_MEMORY )
      S_Coil( "DB2001_MODES_GENERAL".GENERAL.SEMI_SELECTED_MEMORY )
   END_RUNG
   RUNG wire#w3
      Contact( "DB2001_MODES_GENERAL".GENERAL.MANUAL_REQUEST )
      I_Contact( "DB2001_MODES_GENERAL".GENERAL.AUTO_SELECTED_MEMORY )
      I_Contact( "DB2001_MODES_GENERAL".GENERAL.SINGLE_SELECTED_MEMORY )
      I_Contact( "DB2001_MODES_GENERAL".GENERAL.SEMI_SELECTED_MEMORY )
      S_Coil( "DB2001_MODES_GENERAL".GENERAL.MANUAL_SELECTED_MEMORY )
   END_RUNG
   // the same network as SCL:
   #_w1 := #O_BYTE_0.MODE_SELECTED_MEMORY AND ("DB2440_GLOBAL_DATA".GLOBAL_DATA.ANY_MACHINE_CYCLE_RUN OR "DB1101_MACHINE_SEQUENCE".RUNNING) AND NOT "DB2001_MODES_GENERAL".GENERAL.OPTIONS.SGM;
   IF #_w1 AND "DB2001_MODES_GENERAL".GENERAL.AUTOMATIC_REQUEST AND NOT "DB2001_MODES_GENERAL".GENERAL.SINGLE_SELECTED_MEMORY AND NOT "DB2001_MODES_GENERAL".GENERAL.SEMI_SELECTED_MEMORY AND NOT "DB2001_MODES_GENERAL".GENERAL.MANUAL_SELECTED_MEMORY THEN
       "DB2001_MODES_GENERAL".GENERAL.AUTO_SELECTED_MEMORY := TRUE;
   END_IF;
   IF #_w1 AND "DB2001_MODES_GENERAL".GENERAL.SINGLE_REQUEST AND NOT "DB2001_MODES_GENERAL".GENERAL.AUTO_SELECTED_MEMORY AND NOT "DB2001_MODES_GENERAL".GENERAL.SEMI_SELECTED_MEMORY AND NOT "DB2001_MODES_GENERAL".GENERAL.MANUAL_SELECTED_MEMORY THEN
       "DB2001_MODES_GENERAL".GENERAL.SINGLE_SELECTED_MEMORY := TRUE;
   END_IF;
   IF #_w1 AND "DB2001_MODES_GENERAL".GENERAL.SEMIAUTO_REQUEST AND NOT "DB2001_MODES_GENERAL".GENERAL.AUTO_SELECTED_MEMORY AND NOT "DB2001_MODES_GENERAL".GENERAL.SINGLE_SELECTED_MEMORY AND NOT "DB2001_MODES_GENERAL".GENERAL.MANUAL_SELECTED_MEMORY THEN
       "DB2001_MODES_GENERAL".GENERAL.SEMI_SELECTED_MEMORY := TRUE;
   END_IF;
   IF #_w1 AND "DB2001_MODES_GENERAL".GENERAL.MANUAL_REQUEST AND NOT "DB2001_MODES_GENERAL".GENERAL.AUTO_SELECTED_MEMORY AND NOT "DB2001_MODES_GENERAL".GENERAL.SINGLE_SELECTED_MEMORY AND NOT "DB2001_MODES_GENERAL".GENERAL.SEMI_SELECTED_MEMORY THEN
       "DB2001_MODES_GENERAL".GENERAL.MANUAL_SELECTED_MEMORY := TRUE;
   END_IF;
END_REGION

REGION Network 15: CHANGE MODE
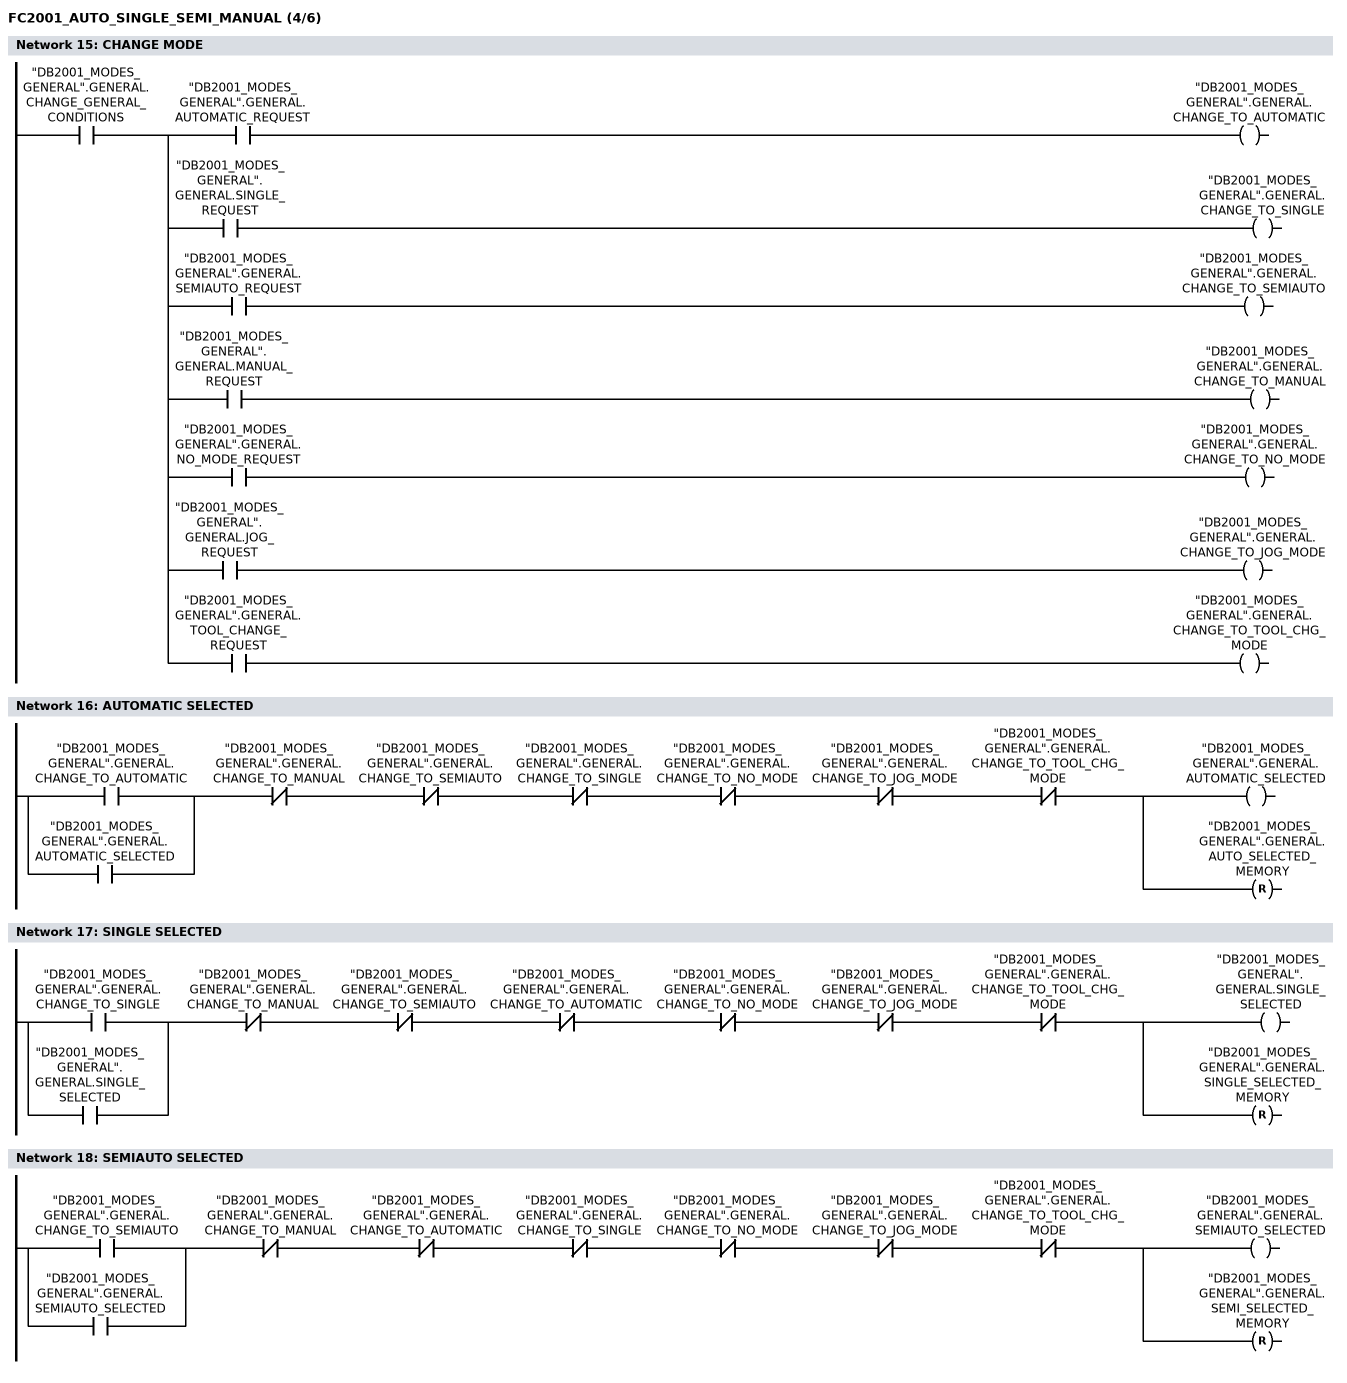
   RUNG wire#powerrail
      Contact( "DB2001_MODES_GENERAL".GENERAL.CHANGE_GENERAL_CONDITIONS )
      wire#w1
      Contact( "DB2001_MODES_GENERAL".GENERAL.AUTOMATIC_REQUEST )
      Coil( "DB2001_MODES_GENERAL".GENERAL.CHANGE_TO_AUTOMATIC )
   END_RUNG
   RUNG wire#w1
      Contact( "DB2001_MODES_GENERAL".GENERAL.SINGLE_REQUEST )
      Coil( "DB2001_MODES_GENERAL".GENERAL.CHANGE_TO_SINGLE )
   END_RUNG
   RUNG wire#w1
      Contact( "DB2001_MODES_GENERAL".GENERAL.SEMIAUTO_REQUEST )
      Coil( "DB2001_MODES_GENERAL".GENERAL.CHANGE_TO_SEMIAUTO )
   END_RUNG
   RUNG wire#w1
      Contact( "DB2001_MODES_GENERAL".GENERAL.MANUAL_REQUEST )
      Coil( "DB2001_MODES_GENERAL".GENERAL.CHANGE_TO_MANUAL )
   END_RUNG
   RUNG wire#w1
      Contact( "DB2001_MODES_GENERAL".GENERAL.NO_MODE_REQUEST )
      Coil( "DB2001_MODES_GENERAL".GENERAL.CHANGE_TO_NO_MODE )
   END_RUNG
   RUNG wire#w1
      Contact( "DB2001_MODES_GENERAL".GENERAL.JOG_REQUEST )
      Coil( "DB2001_MODES_GENERAL".GENERAL.CHANGE_TO_JOG_MODE )
   END_RUNG
   RUNG wire#w1
      Contact( "DB2001_MODES_GENERAL".GENERAL.TOOL_CHANGE_REQUEST )
      Coil( "DB2001_MODES_GENERAL".GENERAL.CHANGE_TO_TOOL_CHG_MODE )
   END_RUNG
   // the same network as SCL:
   "DB2001_MODES_GENERAL".GENERAL.CHANGE_TO_AUTOMATIC := "DB2001_MODES_GENERAL".GENERAL.CHANGE_GENERAL_CONDITIONS AND "DB2001_MODES_GENERAL".GENERAL.AUTOMATIC_REQUEST;
   "DB2001_MODES_GENERAL".GENERAL.CHANGE_TO_SINGLE := "DB2001_MODES_GENERAL".GENERAL.CHANGE_GENERAL_CONDITIONS AND "DB2001_MODES_GENERAL".GENERAL.SINGLE_REQUEST;
   "DB2001_MODES_GENERAL".GENERAL.CHANGE_TO_SEMIAUTO := "DB2001_MODES_GENERAL".GENERAL.CHANGE_GENERAL_CONDITIONS AND "DB2001_MODES_GENERAL".GENERAL.SEMIAUTO_REQUEST;
   "DB2001_MODES_GENERAL".GENERAL.CHANGE_TO_MANUAL := "DB2001_MODES_GENERAL".GENERAL.CHANGE_GENERAL_CONDITIONS AND "DB2001_MODES_GENERAL".GENERAL.MANUAL_REQUEST;
   "DB2001_MODES_GENERAL".GENERAL.CHANGE_TO_NO_MODE := "DB2001_MODES_GENERAL".GENERAL.CHANGE_GENERAL_CONDITIONS AND "DB2001_MODES_GENERAL".GENERAL.NO_MODE_REQUEST;
   "DB2001_MODES_GENERAL".GENERAL.CHANGE_TO_JOG_MODE := "DB2001_MODES_GENERAL".GENERAL.CHANGE_GENERAL_CONDITIONS AND "DB2001_MODES_GENERAL".GENERAL.JOG_REQUEST;
   "DB2001_MODES_GENERAL".GENERAL.CHANGE_TO_TOOL_CHG_MODE := "DB2001_MODES_GENERAL".GENERAL.CHANGE_GENERAL_CONDITIONS AND "DB2001_MODES_GENERAL".GENERAL.TOOL_CHANGE_REQUEST;
END_REGION

REGION Network 16: AUTOMATIC SELECTED
   RUNG wire#powerrail
      Contact( "DB2001_MODES_GENERAL".GENERAL.CHANGE_TO_AUTOMATIC )
      wire#w1
      I_Contact( "DB2001_MODES_GENERAL".GENERAL.CHANGE_TO_MANUAL )
      I_Contact( "DB2001_MODES_GENERAL".GENERAL.CHANGE_TO_SEMIAUTO )
      I_Contact( "DB2001_MODES_GENERAL".GENERAL.CHANGE_TO_SINGLE )
      I_Contact( "DB2001_MODES_GENERAL".GENERAL.CHANGE_TO_NO_MODE )
      I_Contact( "DB2001_MODES_GENERAL".GENERAL.CHANGE_TO_JOG_MODE )
      I_Contact( "DB2001_MODES_GENERAL".GENERAL.CHANGE_TO_TOOL_CHG_MODE )
      wire#w2
      Coil( "DB2001_MODES_GENERAL".GENERAL.AUTOMATIC_SELECTED )
   END_RUNG
   RUNG wire#powerrail
      Contact( "DB2001_MODES_GENERAL".GENERAL.AUTOMATIC_SELECTED )
   END_RUNG wire#w1
   RUNG wire#w2
      R_Coil( "DB2001_MODES_GENERAL".GENERAL.AUTO_SELECTED_MEMORY )
   END_RUNG
   // the same network as SCL:
   "DB2001_MODES_GENERAL".GENERAL.AUTOMATIC_SELECTED := ("DB2001_MODES_GENERAL".GENERAL.CHANGE_TO_AUTOMATIC OR "DB2001_MODES_GENERAL".GENERAL.AUTOMATIC_SELECTED) AND NOT "DB2001_MODES_GENERAL".GENERAL.CHANGE_TO_MANUAL AND NOT "DB2001_MODES_GENERAL".GENERAL.CHANGE_TO_SEMIAUTO AND NOT "DB2001_MODES_GENERAL".GENERAL.CHANGE_TO_SINGLE AND NOT "DB2001_MODES_GENERAL".GENERAL.CHANGE_TO_NO_MODE AND NOT "DB2001_MODES_GENERAL".GENERAL.CHANGE_TO_JOG_MODE AND NOT "DB2001_MODES_GENERAL".GENERAL.CHANGE_TO_TOOL_CHG_MODE;
   IF "DB2001_MODES_GENERAL".GENERAL.AUTOMATIC_SELECTED THEN
       "DB2001_MODES_GENERAL".GENERAL.AUTO_SELECTED_MEMORY := FALSE;
   END_IF;
END_REGION

REGION Network 17: SINGLE SELECTED
   RUNG wire#powerrail
      Contact( "DB2001_MODES_GENERAL".GENERAL.CHANGE_TO_SINGLE )
      wire#w1
      I_Contact( "DB2001_MODES_GENERAL".GENERAL.CHANGE_TO_MANUAL )
      I_Contact( "DB2001_MODES_GENERAL".GENERAL.CHANGE_TO_SEMIAUTO )
      I_Contact( "DB2001_MODES_GENERAL".GENERAL.CHANGE_TO_AUTOMATIC )
      I_Contact( "DB2001_MODES_GENERAL".GENERAL.CHANGE_TO_NO_MODE )
      I_Contact( "DB2001_MODES_GENERAL".GENERAL.CHANGE_TO_JOG_MODE )
      I_Contact( "DB2001_MODES_GENERAL".GENERAL.CHANGE_TO_TOOL_CHG_MODE )
      wire#w2
      Coil( "DB2001_MODES_GENERAL".GENERAL.SINGLE_SELECTED )
   END_RUNG
   RUNG wire#powerrail
      Contact( "DB2001_MODES_GENERAL".GENERAL.SINGLE_SELECTED )
   END_RUNG wire#w1
   RUNG wire#w2
      R_Coil( "DB2001_MODES_GENERAL".GENERAL.SINGLE_SELECTED_MEMORY )
   END_RUNG
   // the same network as SCL:
   "DB2001_MODES_GENERAL".GENERAL.SINGLE_SELECTED := ("DB2001_MODES_GENERAL".GENERAL.CHANGE_TO_SINGLE OR "DB2001_MODES_GENERAL".GENERAL.SINGLE_SELECTED) AND NOT "DB2001_MODES_GENERAL".GENERAL.CHANGE_TO_MANUAL AND NOT "DB2001_MODES_GENERAL".GENERAL.CHANGE_TO_SEMIAUTO AND NOT "DB2001_MODES_GENERAL".GENERAL.CHANGE_TO_AUTOMATIC AND NOT "DB2001_MODES_GENERAL".GENERAL.CHANGE_TO_NO_MODE AND NOT "DB2001_MODES_GENERAL".GENERAL.CHANGE_TO_JOG_MODE AND NOT "DB2001_MODES_GENERAL".GENERAL.CHANGE_TO_TOOL_CHG_MODE;
   IF "DB2001_MODES_GENERAL".GENERAL.SINGLE_SELECTED THEN
       "DB2001_MODES_GENERAL".GENERAL.SINGLE_SELECTED_MEMORY := FALSE;
   END_IF;
END_REGION

REGION Network 18: SEMIAUTO SELECTED
   RUNG wire#powerrail
      Contact( "DB2001_MODES_GENERAL".GENERAL.CHANGE_TO_SEMIAUTO )
      wire#w1
      I_Contact( "DB2001_MODES_GENERAL".GENERAL.CHANGE_TO_MANUAL )
      I_Contact( "DB2001_MODES_GENERAL".GENERAL.CHANGE_TO_AUTOMATIC )
      I_Contact( "DB2001_MODES_GENERAL".GENERAL.CHANGE_TO_SINGLE )
      I_Contact( "DB2001_MODES_GENERAL".GENERAL.CHANGE_TO_NO_MODE )
      I_Contact( "DB2001_MODES_GENERAL".GENERAL.CHANGE_TO_JOG_MODE )
      I_Contact( "DB2001_MODES_GENERAL".GENERAL.CHANGE_TO_TOOL_CHG_MODE )
      wire#w2
      Coil( "DB2001_MODES_GENERAL".GENERAL.SEMIAUTO_SELECTED )
   END_RUNG
   RUNG wire#powerrail
      Contact( "DB2001_MODES_GENERAL".GENERAL.SEMIAUTO_SELECTED )
   END_RUNG wire#w1
   RUNG wire#w2
      R_Coil( "DB2001_MODES_GENERAL".GENERAL.SEMI_SELECTED_MEMORY )
   END_RUNG
   // the same network as SCL:
   "DB2001_MODES_GENERAL".GENERAL.SEMIAUTO_SELECTED := ("DB2001_MODES_GENERAL".GENERAL.CHANGE_TO_SEMIAUTO OR "DB2001_MODES_GENERAL".GENERAL.SEMIAUTO_SELECTED) AND NOT "DB2001_MODES_GENERAL".GENERAL.CHANGE_TO_MANUAL AND NOT "DB2001_MODES_GENERAL".GENERAL.CHANGE_TO_AUTOMATIC AND NOT "DB2001_MODES_GENERAL".GENERAL.CHANGE_TO_SINGLE AND NOT "DB2001_MODES_GENERAL".GENERAL.CHANGE_TO_NO_MODE AND NOT "DB2001_MODES_GENERAL".GENERAL.CHANGE_TO_JOG_MODE AND NOT "DB2001_MODES_GENERAL".GENERAL.CHANGE_TO_TOOL_CHG_MODE;
   IF "DB2001_MODES_GENERAL".GENERAL.SEMIAUTO_SELECTED THEN
       "DB2001_MODES_GENERAL".GENERAL.SEMI_SELECTED_MEMORY := FALSE;
   END_IF;
END_REGION

REGION Network 19: MANUAL SELECTED
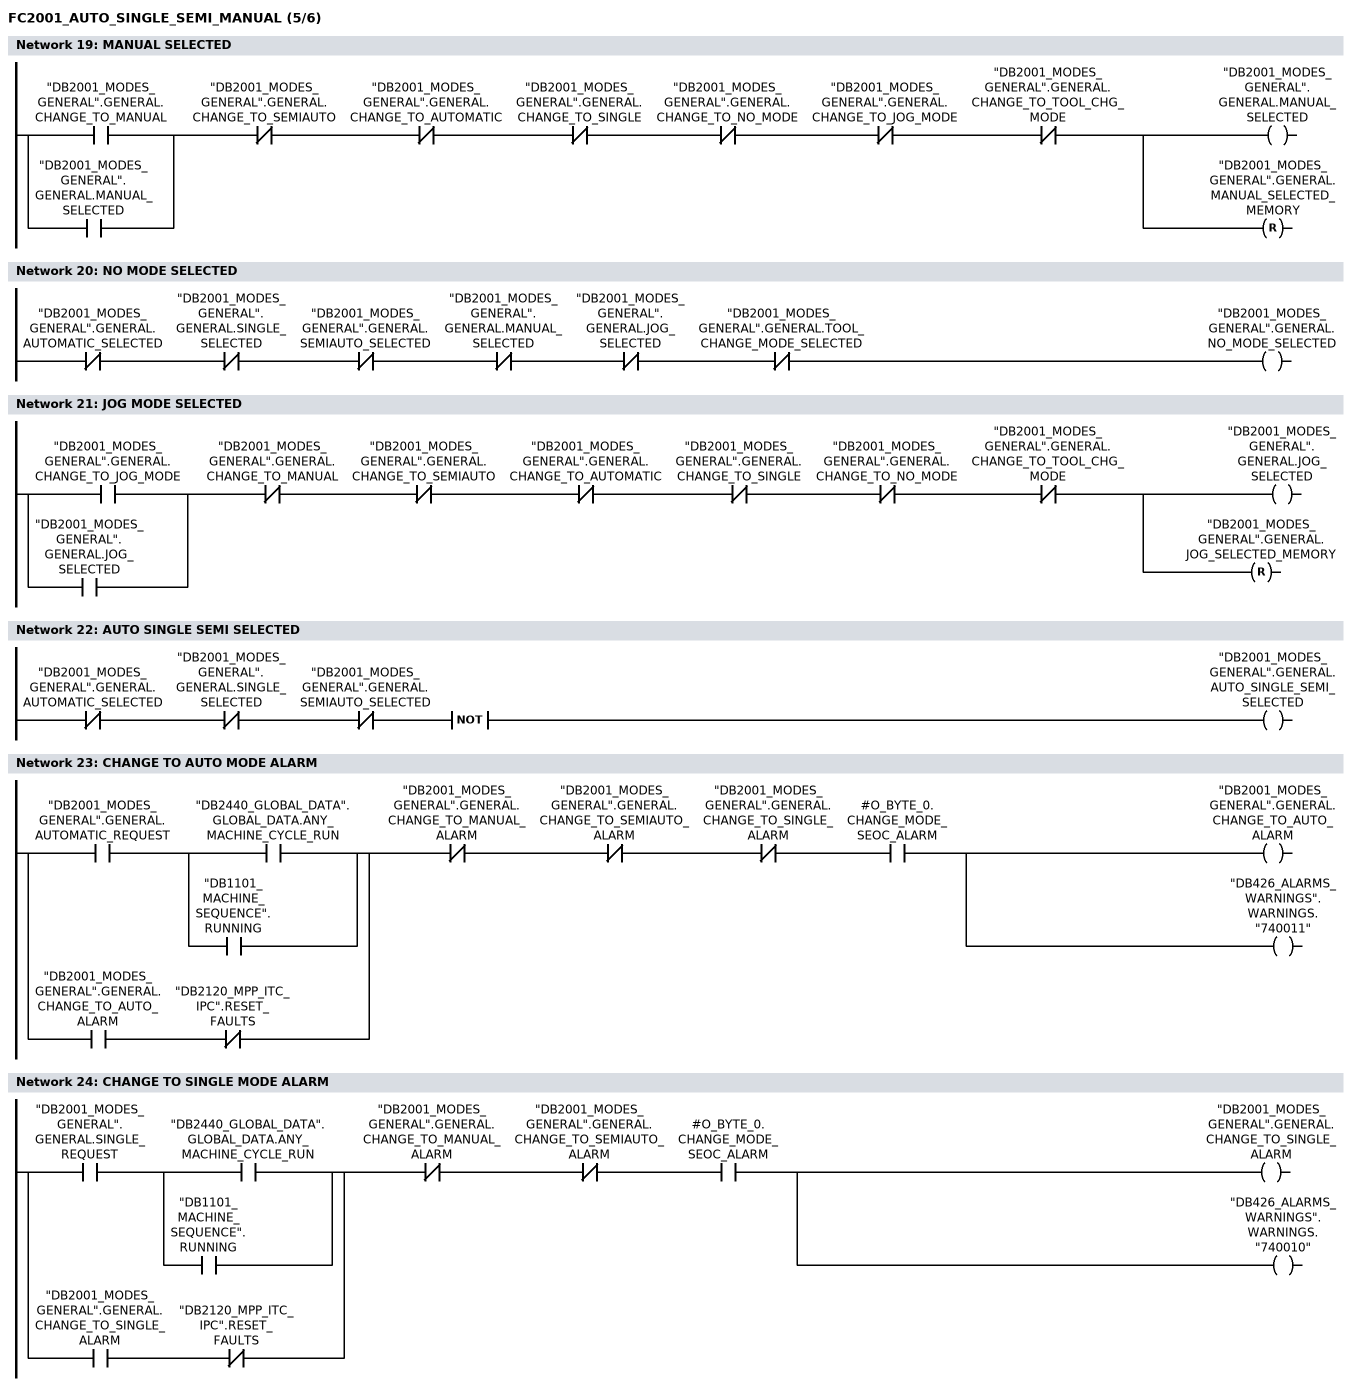
   RUNG wire#powerrail
      Contact( "DB2001_MODES_GENERAL".GENERAL.CHANGE_TO_MANUAL )
      wire#w1
      I_Contact( "DB2001_MODES_GENERAL".GENERAL.CHANGE_TO_SEMIAUTO )
      I_Contact( "DB2001_MODES_GENERAL".GENERAL.CHANGE_TO_AUTOMATIC )
      I_Contact( "DB2001_MODES_GENERAL".GENERAL.CHANGE_TO_SINGLE )
      I_Contact( "DB2001_MODES_GENERAL".GENERAL.CHANGE_TO_NO_MODE )
      I_Contact( "DB2001_MODES_GENERAL".GENERAL.CHANGE_TO_JOG_MODE )
      I_Contact( "DB2001_MODES_GENERAL".GENERAL.CHANGE_TO_TOOL_CHG_MODE )
      wire#w2
      Coil( "DB2001_MODES_GENERAL".GENERAL.MANUAL_SELECTED )
   END_RUNG
   RUNG wire#powerrail
      Contact( "DB2001_MODES_GENERAL".GENERAL.MANUAL_SELECTED )
   END_RUNG wire#w1
   RUNG wire#w2
      R_Coil( "DB2001_MODES_GENERAL".GENERAL.MANUAL_SELECTED_MEMORY )
   END_RUNG
   // the same network as SCL:
   "DB2001_MODES_GENERAL".GENERAL.MANUAL_SELECTED := ("DB2001_MODES_GENERAL".GENERAL.CHANGE_TO_MANUAL OR "DB2001_MODES_GENERAL".GENERAL.MANUAL_SELECTED) AND NOT "DB2001_MODES_GENERAL".GENERAL.CHANGE_TO_SEMIAUTO AND NOT "DB2001_MODES_GENERAL".GENERAL.CHANGE_TO_AUTOMATIC AND NOT "DB2001_MODES_GENERAL".GENERAL.CHANGE_TO_SINGLE AND NOT "DB2001_MODES_GENERAL".GENERAL.CHANGE_TO_NO_MODE AND NOT "DB2001_MODES_GENERAL".GENERAL.CHANGE_TO_JOG_MODE AND NOT "DB2001_MODES_GENERAL".GENERAL.CHANGE_TO_TOOL_CHG_MODE;
   IF "DB2001_MODES_GENERAL".GENERAL.MANUAL_SELECTED THEN
       "DB2001_MODES_GENERAL".GENERAL.MANUAL_SELECTED_MEMORY := FALSE;
   END_IF;
END_REGION

REGION Network 20: NO MODE SELECTED
   RUNG wire#powerrail
      I_Contact( "DB2001_MODES_GENERAL".GENERAL.AUTOMATIC_SELECTED )
      I_Contact( "DB2001_MODES_GENERAL".GENERAL.SINGLE_SELECTED )
      I_Contact( "DB2001_MODES_GENERAL".GENERAL.SEMIAUTO_SELECTED )
      I_Contact( "DB2001_MODES_GENERAL".GENERAL.MANUAL_SELECTED )
      I_Contact( "DB2001_MODES_GENERAL".GENERAL.JOG_SELECTED )
      I_Contact( "DB2001_MODES_GENERAL".GENERAL.TOOL_CHANGE_MODE_SELECTED )
      Coil( "DB2001_MODES_GENERAL".GENERAL.NO_MODE_SELECTED )
   END_RUNG
   // the same network as SCL:
   "DB2001_MODES_GENERAL".GENERAL.NO_MODE_SELECTED := NOT "DB2001_MODES_GENERAL".GENERAL.AUTOMATIC_SELECTED AND NOT "DB2001_MODES_GENERAL".GENERAL.SINGLE_SELECTED AND NOT "DB2001_MODES_GENERAL".GENERAL.SEMIAUTO_SELECTED AND NOT "DB2001_MODES_GENERAL".GENERAL.MANUAL_SELECTED AND NOT "DB2001_MODES_GENERAL".GENERAL.JOG_SELECTED AND NOT "DB2001_MODES_GENERAL".GENERAL.TOOL_CHANGE_MODE_SELECTED;
END_REGION

REGION Network 21: JOG MODE SELECTED
   RUNG wire#powerrail
      Contact( "DB2001_MODES_GENERAL".GENERAL.CHANGE_TO_JOG_MODE )
      wire#w1
      I_Contact( "DB2001_MODES_GENERAL".GENERAL.CHANGE_TO_MANUAL )
      I_Contact( "DB2001_MODES_GENERAL".GENERAL.CHANGE_TO_SEMIAUTO )
      I_Contact( "DB2001_MODES_GENERAL".GENERAL.CHANGE_TO_AUTOMATIC )
      I_Contact( "DB2001_MODES_GENERAL".GENERAL.CHANGE_TO_SINGLE )
      I_Contact( "DB2001_MODES_GENERAL".GENERAL.CHANGE_TO_NO_MODE )
      I_Contact( "DB2001_MODES_GENERAL".GENERAL.CHANGE_TO_TOOL_CHG_MODE )
      wire#w2
      Coil( "DB2001_MODES_GENERAL".GENERAL.JOG_SELECTED )
   END_RUNG
   RUNG wire#powerrail
      Contact( "DB2001_MODES_GENERAL".GENERAL.JOG_SELECTED )
   END_RUNG wire#w1
   RUNG wire#w2
      R_Coil( "DB2001_MODES_GENERAL".GENERAL.JOG_SELECTED_MEMORY )
   END_RUNG
   // the same network as SCL:
   "DB2001_MODES_GENERAL".GENERAL.JOG_SELECTED := ("DB2001_MODES_GENERAL".GENERAL.CHANGE_TO_JOG_MODE OR "DB2001_MODES_GENERAL".GENERAL.JOG_SELECTED) AND NOT "DB2001_MODES_GENERAL".GENERAL.CHANGE_TO_MANUAL AND NOT "DB2001_MODES_GENERAL".GENERAL.CHANGE_TO_SEMIAUTO AND NOT "DB2001_MODES_GENERAL".GENERAL.CHANGE_TO_AUTOMATIC AND NOT "DB2001_MODES_GENERAL".GENERAL.CHANGE_TO_SINGLE AND NOT "DB2001_MODES_GENERAL".GENERAL.CHANGE_TO_NO_MODE AND NOT "DB2001_MODES_GENERAL".GENERAL.CHANGE_TO_TOOL_CHG_MODE;
   IF "DB2001_MODES_GENERAL".GENERAL.JOG_SELECTED THEN
       "DB2001_MODES_GENERAL".GENERAL.JOG_SELECTED_MEMORY := FALSE;
   END_IF;
END_REGION

REGION Network 22: AUTO SINGLE SEMI SELECTED
   RUNG wire#powerrail
      I_Contact( "DB2001_MODES_GENERAL".GENERAL.AUTOMATIC_SELECTED )
      I_Contact( "DB2001_MODES_GENERAL".GENERAL.SINGLE_SELECTED )
      I_Contact( "DB2001_MODES_GENERAL".GENERAL.SEMIAUTO_SELECTED )
      Not()
      Coil( "DB2001_MODES_GENERAL".GENERAL.AUTO_SINGLE_SEMI_SELECTED )
   END_RUNG
   // the same network as SCL:
   "DB2001_MODES_GENERAL".GENERAL.AUTO_SINGLE_SEMI_SELECTED := NOT (NOT "DB2001_MODES_GENERAL".GENERAL.AUTOMATIC_SELECTED AND NOT "DB2001_MODES_GENERAL".GENERAL.SINGLE_SELECTED AND NOT "DB2001_MODES_GENERAL".GENERAL.SEMIAUTO_SELECTED);
END_REGION

REGION Network 23: CHANGE TO AUTO MODE ALARM
   RUNG wire#powerrail
      Contact( "DB2001_MODES_GENERAL".GENERAL.AUTOMATIC_REQUEST )
      wire#w1
      Contact( "DB2440_GLOBAL_DATA".GLOBAL_DATA.ANY_MACHINE_CYCLE_RUN )
      wire#w2
      I_Contact( "DB2001_MODES_GENERAL".GENERAL.CHANGE_TO_MANUAL_ALARM )
      I_Contact( "DB2001_MODES_GENERAL".GENERAL.CHANGE_TO_SEMIAUTO_ALARM )
      I_Contact( "DB2001_MODES_GENERAL".GENERAL.CHANGE_TO_SINGLE_ALARM )
      Contact( #O_BYTE_0.CHANGE_MODE_SEOC_ALARM )
      wire#w3
      Coil( "DB2001_MODES_GENERAL".GENERAL.CHANGE_TO_AUTO_ALARM )
   END_RUNG
   RUNG wire#w1
      Contact( "DB1101_MACHINE_SEQUENCE".RUNNING )
   END_RUNG wire#w2
   RUNG wire#powerrail
      Contact( "DB2001_MODES_GENERAL".GENERAL.CHANGE_TO_AUTO_ALARM )
      I_Contact( "DB2120_MPP_ITC_IPC".RESET_FAULTS )
   END_RUNG wire#w2
   RUNG wire#w3
      Coil( "DB426_ALARMS_WARNINGS".WARNINGS."740011" )
   END_RUNG
   // the same network as SCL:
   "DB2001_MODES_GENERAL".GENERAL.CHANGE_TO_AUTO_ALARM := (("DB2001_MODES_GENERAL".GENERAL.AUTOMATIC_REQUEST AND ("DB2440_GLOBAL_DATA".GLOBAL_DATA.ANY_MACHINE_CYCLE_RUN OR "DB1101_MACHINE_SEQUENCE".RUNNING)) OR ("DB2001_MODES_GENERAL".GENERAL.CHANGE_TO_AUTO_ALARM AND NOT "DB2120_MPP_ITC_IPC".RESET_FAULTS)) AND NOT "DB2001_MODES_GENERAL".GENERAL.CHANGE_TO_MANUAL_ALARM AND NOT "DB2001_MODES_GENERAL".GENERAL.CHANGE_TO_SEMIAUTO_ALARM AND NOT "DB2001_MODES_GENERAL".GENERAL.CHANGE_TO_SINGLE_ALARM AND #O_BYTE_0.CHANGE_MODE_SEOC_ALARM;
   "DB426_ALARMS_WARNINGS".WARNINGS."740011" := "DB2001_MODES_GENERAL".GENERAL.CHANGE_TO_AUTO_ALARM;
END_REGION

REGION Network 24: CHANGE TO SINGLE MODE ALARM
   RUNG wire#powerrail
      Contact( "DB2001_MODES_GENERAL".GENERAL.SINGLE_REQUEST )
      wire#w1
      Contact( "DB2440_GLOBAL_DATA".GLOBAL_DATA.ANY_MACHINE_CYCLE_RUN )
      wire#w2
      I_Contact( "DB2001_MODES_GENERAL".GENERAL.CHANGE_TO_MANUAL_ALARM )
      I_Contact( "DB2001_MODES_GENERAL".GENERAL.CHANGE_TO_SEMIAUTO_ALARM )
      Contact( #O_BYTE_0.CHANGE_MODE_SEOC_ALARM )
      wire#w3
      Coil( "DB2001_MODES_GENERAL".GENERAL.CHANGE_TO_SINGLE_ALARM )
   END_RUNG
   RUNG wire#w1
      Contact( "DB1101_MACHINE_SEQUENCE".RUNNING )
   END_RUNG wire#w2
   RUNG wire#powerrail
      Contact( "DB2001_MODES_GENERAL".GENERAL.CHANGE_TO_SINGLE_ALARM )
      I_Contact( "DB2120_MPP_ITC_IPC".RESET_FAULTS )
   END_RUNG wire#w2
   RUNG wire#w3
      Coil( "DB426_ALARMS_WARNINGS".WARNINGS."740010" )
   END_RUNG
   // the same network as SCL:
   "DB2001_MODES_GENERAL".GENERAL.CHANGE_TO_SINGLE_ALARM := (("DB2001_MODES_GENERAL".GENERAL.SINGLE_REQUEST AND ("DB2440_GLOBAL_DATA".GLOBAL_DATA.ANY_MACHINE_CYCLE_RUN OR "DB1101_MACHINE_SEQUENCE".RUNNING)) OR ("DB2001_MODES_GENERAL".GENERAL.CHANGE_TO_SINGLE_ALARM AND NOT "DB2120_MPP_ITC_IPC".RESET_FAULTS)) AND NOT "DB2001_MODES_GENERAL".GENERAL.CHANGE_TO_MANUAL_ALARM AND NOT "DB2001_MODES_GENERAL".GENERAL.CHANGE_TO_SEMIAUTO_ALARM AND #O_BYTE_0.CHANGE_MODE_SEOC_ALARM;
   "DB426_ALARMS_WARNINGS".WARNINGS."740010" := "DB2001_MODES_GENERAL".GENERAL.CHANGE_TO_SINGLE_ALARM;
END_REGION

REGION Network 25: CHANGE TO SEMIAUTO MODE ALARM
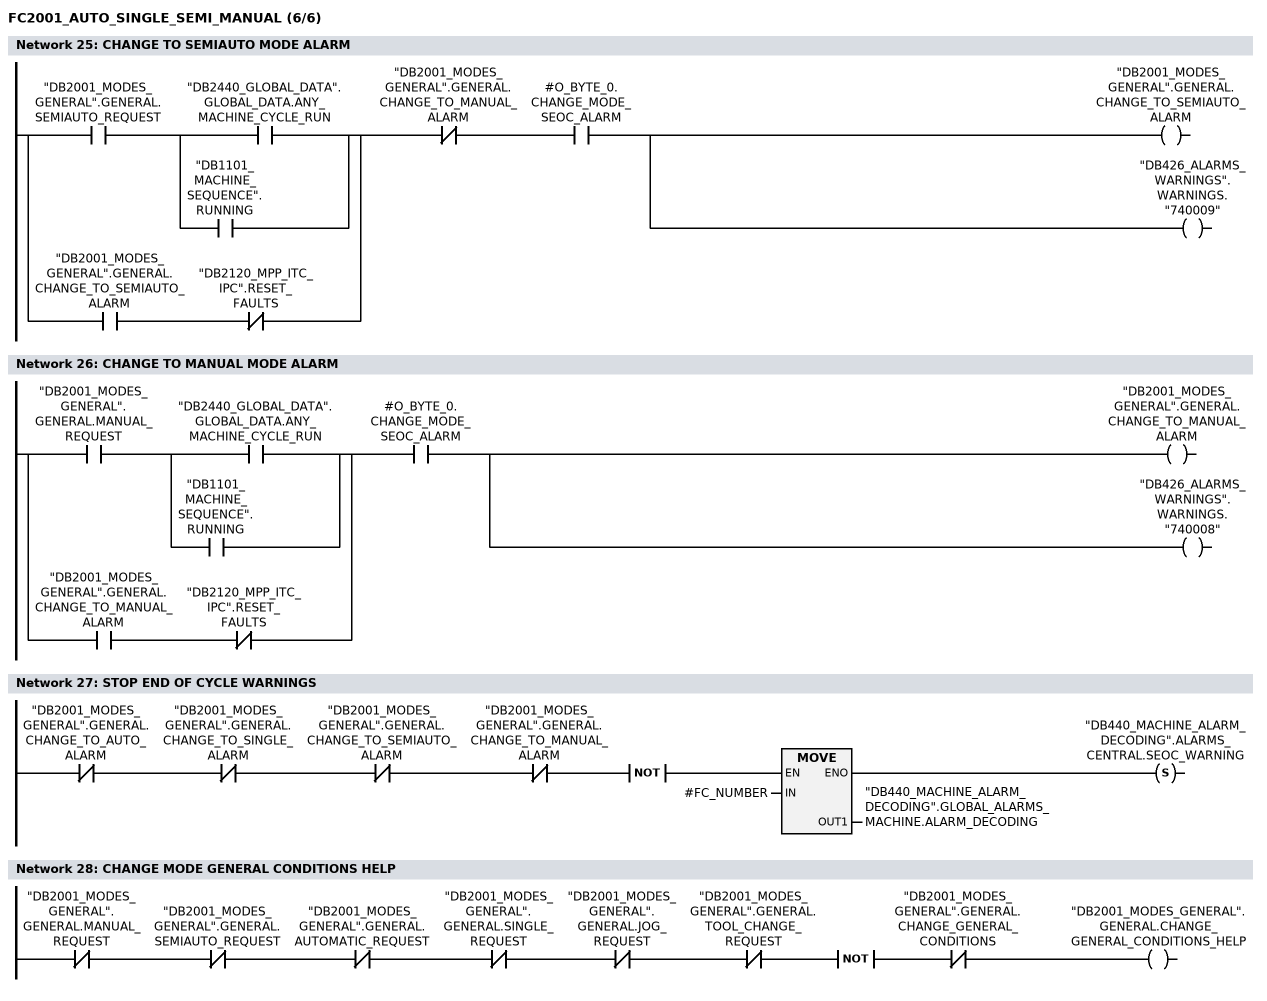
   RUNG wire#powerrail
      Contact( "DB2001_MODES_GENERAL".GENERAL.SEMIAUTO_REQUEST )
      wire#w1
      Contact( "DB2440_GLOBAL_DATA".GLOBAL_DATA.ANY_MACHINE_CYCLE_RUN )
      wire#w2
      I_Contact( "DB2001_MODES_GENERAL".GENERAL.CHANGE_TO_MANUAL_ALARM )
      Contact( #O_BYTE_0.CHANGE_MODE_SEOC_ALARM )
      wire#w3
      Coil( "DB2001_MODES_GENERAL".GENERAL.CHANGE_TO_SEMIAUTO_ALARM )
   END_RUNG
   RUNG wire#w1
      Contact( "DB1101_MACHINE_SEQUENCE".RUNNING )
   END_RUNG wire#w2
   RUNG wire#powerrail
      Contact( "DB2001_MODES_GENERAL".GENERAL.CHANGE_TO_SEMIAUTO_ALARM )
      I_Contact( "DB2120_MPP_ITC_IPC".RESET_FAULTS )
   END_RUNG wire#w2
   RUNG wire#w3
      Coil( "DB426_ALARMS_WARNINGS".WARNINGS."740009" )
   END_RUNG
   // the same network as SCL:
   "DB2001_MODES_GENERAL".GENERAL.CHANGE_TO_SEMIAUTO_ALARM := (("DB2001_MODES_GENERAL".GENERAL.SEMIAUTO_REQUEST AND ("DB2440_GLOBAL_DATA".GLOBAL_DATA.ANY_MACHINE_CYCLE_RUN OR "DB1101_MACHINE_SEQUENCE".RUNNING)) OR ("DB2001_MODES_GENERAL".GENERAL.CHANGE_TO_SEMIAUTO_ALARM AND NOT "DB2120_MPP_ITC_IPC".RESET_FAULTS)) AND NOT "DB2001_MODES_GENERAL".GENERAL.CHANGE_TO_MANUAL_ALARM AND #O_BYTE_0.CHANGE_MODE_SEOC_ALARM;
   "DB426_ALARMS_WARNINGS".WARNINGS."740009" := "DB2001_MODES_GENERAL".GENERAL.CHANGE_TO_SEMIAUTO_ALARM;
END_REGION

REGION Network 26: CHANGE TO MANUAL MODE ALARM
   RUNG wire#powerrail
      Contact( "DB2001_MODES_GENERAL".GENERAL.MANUAL_REQUEST )
      wire#w1
      Contact( "DB2440_GLOBAL_DATA".GLOBAL_DATA.ANY_MACHINE_CYCLE_RUN )
      wire#w2
      Contact( #O_BYTE_0.CHANGE_MODE_SEOC_ALARM )
      wire#w3
      Coil( "DB2001_MODES_GENERAL".GENERAL.CHANGE_TO_MANUAL_ALARM )
   END_RUNG
   RUNG wire#w1
      Contact( "DB1101_MACHINE_SEQUENCE".RUNNING )
   END_RUNG wire#w2
   RUNG wire#powerrail
      Contact( "DB2001_MODES_GENERAL".GENERAL.CHANGE_TO_MANUAL_ALARM )
      I_Contact( "DB2120_MPP_ITC_IPC".RESET_FAULTS )
   END_RUNG wire#w2
   RUNG wire#w3
      Coil( "DB426_ALARMS_WARNINGS".WARNINGS."740008" )
   END_RUNG
   // the same network as SCL:
   "DB2001_MODES_GENERAL".GENERAL.CHANGE_TO_MANUAL_ALARM := (("DB2001_MODES_GENERAL".GENERAL.MANUAL_REQUEST AND ("DB2440_GLOBAL_DATA".GLOBAL_DATA.ANY_MACHINE_CYCLE_RUN OR "DB1101_MACHINE_SEQUENCE".RUNNING)) OR ("DB2001_MODES_GENERAL".GENERAL.CHANGE_TO_MANUAL_ALARM AND NOT "DB2120_MPP_ITC_IPC".RESET_FAULTS)) AND #O_BYTE_0.CHANGE_MODE_SEOC_ALARM;
   "DB426_ALARMS_WARNINGS".WARNINGS."740008" := "DB2001_MODES_GENERAL".GENERAL.CHANGE_TO_MANUAL_ALARM;
END_REGION

REGION Network 27: STOP END OF CYCLE WARNINGS
   RUNG wire#powerrail
      I_Contact( "DB2001_MODES_GENERAL".GENERAL.CHANGE_TO_AUTO_ALARM )
      I_Contact( "DB2001_MODES_GENERAL".GENERAL.CHANGE_TO_SINGLE_ALARM )
      I_Contact( "DB2001_MODES_GENERAL".GENERAL.CHANGE_TO_SEMIAUTO_ALARM )
      I_Contact( "DB2001_MODES_GENERAL".GENERAL.CHANGE_TO_MANUAL_ALARM )
      Not()
      { S7_GenerateENO := "TRUE" } Move(in := #FC_NUMBER, out1 => "DB440_MACHINE_ALARM_DECODING".GLOBAL_ALARMS_MACHINE.ALARM_DECODING)
      S_Coil( "DB440_MACHINE_ALARM_DECODING".ALARMS_CENTRAL.SEOC_WARNING )
   END_RUNG
   // the same network as SCL:
   // ENO of a box is taken as its EN; it also drops when the box reports an error
   IF NOT (NOT "DB2001_MODES_GENERAL".GENERAL.CHANGE_TO_AUTO_ALARM AND NOT "DB2001_MODES_GENERAL".GENERAL.CHANGE_TO_SINGLE_ALARM AND NOT "DB2001_MODES_GENERAL".GENERAL.CHANGE_TO_SEMIAUTO_ALARM AND NOT "DB2001_MODES_GENERAL".GENERAL.CHANGE_TO_MANUAL_ALARM) THEN
       "DB440_MACHINE_ALARM_DECODING".GLOBAL_ALARMS_MACHINE.ALARM_DECODING := #FC_NUMBER;
       "DB440_MACHINE_ALARM_DECODING".ALARMS_CENTRAL.SEOC_WARNING := TRUE;
   END_IF;
END_REGION

REGION Network 28: CHANGE MODE GENERAL CONDITIONS HELP
   RUNG wire#powerrail
      I_Contact( "DB2001_MODES_GENERAL".GENERAL.MANUAL_REQUEST )
      I_Contact( "DB2001_MODES_GENERAL".GENERAL.SEMIAUTO_REQUEST )
      I_Contact( "DB2001_MODES_GENERAL".GENERAL.AUTOMATIC_REQUEST )
      I_Contact( "DB2001_MODES_GENERAL".GENERAL.SINGLE_REQUEST )
      I_Contact( "DB2001_MODES_GENERAL".GENERAL.JOG_REQUEST )
      I_Contact( "DB2001_MODES_GENERAL".GENERAL.TOOL_CHANGE_REQUEST )
      Not()
      I_Contact( "DB2001_MODES_GENERAL".GENERAL.CHANGE_GENERAL_CONDITIONS )
      Coil( "DB2001_MODES_GENERAL".GENERAL.CHANGE_GENERAL_CONDITIONS_HELP )
   END_RUNG
   // the same network as SCL:
   "DB2001_MODES_GENERAL".GENERAL.CHANGE_GENERAL_CONDITIONS_HELP := NOT (NOT "DB2001_MODES_GENERAL".GENERAL.MANUAL_REQUEST AND NOT "DB2001_MODES_GENERAL".GENERAL.SEMIAUTO_REQUEST AND NOT "DB2001_MODES_GENERAL".GENERAL.AUTOMATIC_REQUEST AND NOT "DB2001_MODES_GENERAL".GENERAL.SINGLE_REQUEST AND NOT "DB2001_MODES_GENERAL".GENERAL.JOG_REQUEST AND NOT "DB2001_MODES_GENERAL".GENERAL.TOOL_CHANGE_REQUEST) AND NOT "DB2001_MODES_GENERAL".GENERAL.CHANGE_GENERAL_CONDITIONS;
END_REGION
END_FUNCTION
